PROGRAM pouEtherCATdiag
VAR
	iVal: WORD;
	tVal: WORD;
	tmask: WORD;
	state: UINT;
	i: UINT;
END_VAR

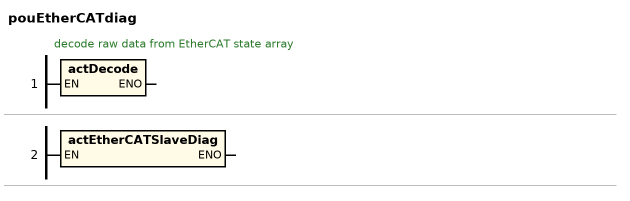
// NETWORK 1
// decode raw data from EtherCAT state array
actDecode();

// NETWORK 2
actEtherCATSlaveDiag();

ACTION actDecode:
///EtherCAT state decoding

//0x___1 = Slave in 'INIT' state
//0x___2 = Slave in 'PREOP' state
//0x___3 = Slave in 'BOOT' state
//0x___4 = Slave in 'SAFEOP' state
//0x___8 = Slave in 'OP' state

tVal := iVal AND 16#000F;

	//from the control word, colour the box
	CASE tVal OF 
 		16#0001 : state := 1;// Slave in 'INIT' state
		16#0002 : state := 2;// Slave in 'PREOP' state
		16#0003 : state := 3;//	Slave in 'BOOT' state
		16#0004 : state := 4;// Slave in 'SAFEOP' state
		16#0008 : state := 5;//	Slave in 'OP' state	: 	profibusDiag.DPslaveDiag[i].currentState := HMIColour.colourRed;
			
	ELSE 
			//invalid state
			state:= 99;
	END_CASE;
		
	//move state into correct area
	etherCATdiag.ethercatdiagtest.currentState.state := state;
 
	//0x001_ = Slave signals error
	//0x002_ = Invalid vendorId, productCode... read
	//0x004_ = Initialization error occurred
	//0x008_ = Slave disabled
	//0x010_ = Slave not present
	//0x020_ = Slave signals link error
	//0x040_ = Slave signals missing link
	//0x080_ = Slave signals unexpected link
	//0x100_ = Communication port A
	//0x200_ = Communication port B
	//0x400_ = Communication port C
	//0x800_ = Communication port D


tVal := iVal AND 16#FFF0;
	//from the control word, colour the box
	CASE tVal OF 
		16#001 : state := 1;		//Slave signals error
		16#002 : state := 2;		//Invalid vendorId, productCode... read
		16#008 : state := 3;		//Slave disabled
		16#010 : state := 4;		//Slave NOT present
		16#020 : state := 5;		//Slave signals link error
		16#040 : state := 6;		//Slave signals missing link
		16#080 : state := 7;		//Slave signals unexpected link
		16#100 : state := 8;		//Communication port A
		16#200 : state := 9;		//Communication port B
		16#400 : state := 10;		//Communication port C
		16#800 : state := 11;		//Communication port D	
	ELSE 
			//invalid state
			state:= 99;
	END_CASE;


	//move state into correct area
	etherCATdiag.ethercatdiagtest.currentState.suffix := state;
END_ACTION

ACTION actEtherCATSlaveDiag:
FOR i := 1 TO etherCATdiag.maxNumEtherCATSlaves DO
	
	//check values for fault
	//current state
	IF etherCATdiag.EtherCATslaveDiag[i].currentState.state <> EtherCATstate.OP OR
		etherCATdiag.EtherCATslaveDiag[i].currentState.suffix <> EtherCATSuffix.NoState THEN
		etherCATdiag.EtherCATslaveDiag[i].currentState.isFault := TRUE;
		ELSE
		etherCATdiag.EtherCATslaveDiag[i].currentState.isFault := FALSE;	
	END_IF
	

	//record outer box
	//record previous state, latching 
	IF etherCATdiag.EtherCATslaveDiag[i].currentState.isFault = FALSE AND 
	   etherCATdiag.EtherCATslaveDiag[i].historicalState.isFault = FALSE THEN
		//at this time, record the current state in the historical state
		etherCATdiag.EtherCATslaveDiag[i].historicalState.state := etherCATdiag.EtherCATslaveDiag[i].currentState.state;
		etherCATdiag.EtherCATslaveDiag[i].historicalState.suffix := etherCATdiag.EtherCATslaveDiag[i].currentState.suffix;
	END_IF
	
	//clear inner box when fault is resolved
	IF 	etherCATdiag.EtherCATslaveDiag[i].currentState.isFault = FALSE AND
	   HMIData.btnReset THEN
	   etherCATdiag.EtherCATslaveDiag[i].historicalState.isFault := FALSE;
	END_IF
	
	
			//check if any suffix fault exits
			IF etherCATdiag.EtherCATslaveDiag[i].currentState.suffix THEN
				
				//check suffix
				CASE etherCATdiag.EtherCATslaveDiag[i].currentState.suffix OF 
				EtherCATSuffix.SSError						: 	etherCATdiag.EtherCATslaveDiag[i].currentState.colour := HMIColour.colourRed;
				EtherCATSuffix.InvalidVendor				: 	etherCATdiag.EtherCATslaveDiag[i].currentState.colour := HMIColour.colourRed;
				EtherCATSuffix.InitError 					: 	etherCATdiag.EtherCATslaveDiag[i].currentState.colour := HMIColour.colourRed;
				EtherCATSuffix.SlaveDisabled				:	etherCATdiag.EtherCATslaveDiag[i].currentState.colour := HMIColour.colourRed;
				EtherCATSuffix.SlaveNotPresent				: 	etherCATdiag.EtherCATslaveDiag[i].currentState.colour := HMIColour.colourRed;
				EtherCATSuffix.SlaveSignalsLinkError		:	etherCATdiag.EtherCATslaveDiag[i].currentState.colour := HMIColour.colourRed;
				EtherCATSuffix.SlaveSignalsMissingLink		:	etherCATdiag.EtherCATslaveDiag[i].currentState.colour := HMIColour.colourRed;
				EtherCATSuffix.SlaveSignalsUnExpectLink		:	etherCATdiag.EtherCATslaveDiag[i].currentState.colour := HMIColour.colourRed;
				EtherCATSuffix.CommsPortA					:	etherCATdiag.EtherCATslaveDiag[i].currentState.colour := HMIColour.colourRed;
				EtherCATSuffix.CommsPortB					:	etherCATdiag.EtherCATslaveDiag[i].currentState.colour := HMIColour.colourRed;
				EtherCATSuffix.CommsPortC					:	etherCATdiag.EtherCATslaveDiag[i].currentState.colour := HMIColour.colourRed;
				EtherCATSuffix.CommsPortD					:	etherCATdiag.EtherCATslaveDiag[i].currentState.colour := HMIColour.colourRed;
				END_CASE;
				
			ELSE
				//otherwise check state to get green
				CASE etherCATdiag.EtherCATslaveDiag[i].currentState.state OF 
				EtherCATstate.INIT		: 	etherCATdiag.EtherCATslaveDiag[i].currentState.colour := HMIColour.colourRed;
				EtherCATstate.PREOP		: 	etherCATdiag.EtherCATslaveDiag[i].currentState.colour := HMIColour.colourRed;
				EtherCATstate.BOOT		: 	etherCATdiag.EtherCATslaveDiag[i].currentState.colour := HMIColour.colourRed;
				EtherCATstate.SAFEOP	: 	etherCATdiag.EtherCATslaveDiag[i].currentState.colour := HMIColour.colourRed;
				EtherCATstate.OP		: 	etherCATdiag.EtherCATslaveDiag[i].currentState.colour := HMIColour.colourGreen;
				END_CASE;
				
			END_IF
	
	
	
	
END_FOR
END_ACTION

END_PROGRAM

(* stored: Version 1.1.0.1, ProductVersion 3.1.4024.12
   POU pouEtherCATdiag: Id {73650198-8c30-49b6-b422-2b646bfaa17e}, SpecialFunc None
   Action actDecode: Id {f7267f8b-08d5-4b9b-952d-81dcefa7c961}
   Action actEtherCATSlaveDiag: Id {ad26e273-933b-4a92-8e3a-4cf2719bddff} *)
